(* Logix 5000 project; controller SRP_BullPMM_TestBench_V1 vendor 1 type 14 code 77 rev 20.11; software revision 20.05 *)

TASK MainTask (continuous, watchdog 500 ms) : MainProgram

MODULES
   Controller : vendor 1 type 14 code 77 (CompactLogixL32EController 0, rev 20.11)
      LocalENB : 1769-L32E Ethernet Port (CompactLogixL32Ethernet 1, rev 20.11)
         VSD_DC : vendor 1 type 123 code 121 (Ethernet 192.168.2.130, rev 5.6, Output RPI 20 ms)
             : vendor 1 type 123 code 8192 (DPI 5, rev 4.1)
      Local : CompactBus (CompactVirtualAdapter 3, rev 20.11)
END_MODULES

VAR_GLOBAL   (* controller tags *)
   CTU_SRPSim : COUNTER := (PRE := 280, ACC := 248);
   CurrentLimitLocal : INT;
   DC_CommandOFF : BOOL;
   DC_CommandON : BOOL;
   DC_CommandReset : BOOL;
   DC_CommandSpeed : INT;
   DC_CurrentLimit : INT;
   DC_LoadSent : INT := 7;
   DC_MaxLoad : REAL := 15.0;
   DC_MinLoad : REAL := 3.0;
   DC_OutputPower : REAL;
   DC_OutputVoltage : REAL;
   DC_RPMFeedback : INT := -22;
   DC_RPMReference : DINT := 100;
   DC_SpeedReference : INT := 140;
   DC_Timer_OFF : TIMER := (PRE := 1000);
   DC_Timer_ON : TIMER := (PRE := 1000);
   DC_Timer_RST : TIMER := (PRE := 1000);
   habilitado : BOOL; {access Read Only}
   Samples : INT := 280;
   SPM : REAL := 8.51;
   SRP_Displacement : REAL[400] := ([0] := 4.0, [1] := 1.0, [2] := 2.0, [3] := 3.0, [4] := 4.0, [5] := 5.0, [6] := 6.0, [7] := 7.0, [8] := 8.0, [9] := 9.0, [10] := 10.0, [11] := 11.0, [12] := 12.0, [13] := 13.0, [14] := 14.0, [15] := 15.0, [16] := 16.0, [17] := 17.0, [18] := 18.0, [19] := 19.0, [20] := 20.0, [21] := 21.0, [22] := 22.0, [23] := 23.0, [24] := 24.0, [25] := 25.0, [26] := 26.0, [27] := 27.0, [28] := 28.0, [29] := 29.0, [30] := 30.0, [31] := 31.0, [32] := 32.0, [33] := 33.0, [34] := 34.0, [35] := 35.0, [36] := 36.0, [37] := 37.0, [38] := 38.0, [39] := 39.0, [40] := 40.0, [41] := 41.0, [42] := 42.0, [43] := 43.0, [44] := 44.0, [45] := 45.0, [46] := 46.0, [47] := 47.0, [48] := 48.0, [49] := 49.0, [50] := 50.0, [51] := 51.0, [52] := 52.0, [53] := 53.0, [54] := 54.0, [55] := 55.0, [56] := 56.0, [57] := 57.0, [58] := 58.0, [59] := 59.0,
        [60] := 60.0, [61] := 61.0, [62] := 62.0, [63] := 63.0, [64] := 64.0, [65] := 65.0, [66] := 66.0, [67] := 67.0, [68] := 68.0, [69] := 69.0, [70] := 70.0, [71] := 71.0, [72] := 72.0, [73] := 73.0, [74] := 74.0, [75] := 75.0, [76] := 76.0, [77] := 77.0, [78] := 78.0, [79] := 79.0, [80] := 80.0, [81] := 81.0, [82] := 82.0, [83] := 83.0, [84] := 84.0, [85] := 85.0, [86] := 86.0, [87] := 87.0, [88] := 88.0, [89] := 89.0, [90] := 90.0, [91] := 91.0, [92] := 92.0, [93] := 93.0, [94] := 94.0, [95] := 95.0, [96] := 96.0, [97] := 97.0, [98] := 98.0, [99] := 99.0, [100] := 100.0, [101] := 101.0, [102] := 102.0, [103] := 103.0, [104] := 104.0, [105] := 105.0, [106] := 106.0, [107] := 107.0, [108] := 108.0, [109] := 109.0, [110] := 110.0, [111] := 111.0, [112] := 112.0, [113] := 113.0, [114] := 114.0, [115] := 115.0, [116] := 116.0, [117] := 117.0, [118] := 118.0, [119] := 119.0,
        [120] := 120.0, [121] := 121.0, [122] := 122.0, [123] := 123.0, [124] := 124.0, [125] := 125.0, [126] := 126.0, [127] := 127.0, [128] := 128.0, [129] := 129.0, [130] := 130.0, [131] := 131.0, [132] := 132.0, [133] := 133.0, [134] := 134.0, [135] := 135.0, [136] := 136.0, [137] := 137.0, [138] := 138.0, [139] := 139.0, [140] := 140.0); {access Read Only}
   SRP_Displacement_actual : REAL := 34.528854; {produced, access Read Only}
   SRP_Load : REAL[400] := ([1] := 12.0, [2] := 5.0, [3] := 6.0, [4] := 7.0, [5] := 89.0, [6] := 9.0, [7] := 3.0, [8] := 4.0, [9] := 6.0, [12] := 8.0, [14] := 56.0, [16] := 56.0, [18] := 56.0, [21] := 8765.0, [24] := 5678.0, [26] := 5678.0, [27] := 567.0, [28] := 8.0, [29] := 324.0, [31] := 234.0, [32] := 324.0, [33] := 234.0, [34] := 234.0, [35] := 342.0, [36] := 34.0, [43] := 432.0, [45] := 4.0, [46] := 4.0, [47] := 4.0, [48] := 4.0, [50] := 3.0, [52] := 2.0, [55] := 245.0, [56] := 2345.0, [57] := 2345.0, [58] := 724.0, [59] := 4325.0, [60] := 3245.0, [61] := 2345.0, [86] := 2345.0, [89] := 2345.0, [91] := 2345.0, [92] := 2345.0, [98] := 234.0, [99] := 4.0, [100] := 2.0, [101] := 3.0, [102] := 45.0, [103] := 2345.0, [104] := 2345.0, [105] := 5234.0, [106] := 354.0, [170] := 123.0, [191] := 345.0, [215] := 132.0, [216] := 5.0, [217] := 6.0, [219] := 8.0, [220] := 435.0, [221] := 34.0,
        [222] := 34.0, [223] := 3.0, [226] := 234.0, [227] := 3.0, [228] := 456.0, [231] := 546.0, [232] := 543.0, [233] := 453.0, [234] := 543.0, [235] := 34.0, [236] := 4.0, [294] := 4234.0, [295] := 3.0, [296] := 34.0, [297] := 4334.0, [298] := 34.0, [299] := 34.0, [300] := 43.0, [301] := 34.0, [303] := 1234.0); {access Read Only}
   SRP_Load_Actual : REAL := 8.460728; {produced, access Read Only}
   SRP_LoadEXC : REAL[400] := ([0] := 9.395175, [1] := 9.461731, [2] := 9.6614, [3] := 9.7812, [4] := 9.741267, [5] := 9.711983, [6] := 9.703996, [7] := 9.725293, [8] := 9.805161, [9] := 9.842433, [10] := 9.794512, [11] := 9.749254, [12] := 9.70932, [13] := 9.69601, [14] := 9.735943, [15] := 9.7306185, [16] := 9.634778, [17] := 9.586858, [18] := 9.634777, [19] := 9.751916, [20] := 10.007491, [21] := 10.223133, [22] := 10.358908, [23] := 10.473384, [24] := 10.545264, [25] := 10.633119, [26] := 10.752919, [27] := 10.856748, [28] := 10.928628, [29] := 11.029794, [30] := 11.109661, [31] := 11.220809, [32] := 11.347599, [33] := 11.419147, [34] := 11.463074, [35] := 11.515653, [36] := 11.572558, [37] := 11.655421, [38] := 11.751262, [39] := 11.805838, [40] := 11.839782, [41] := 11.900348, [42] := 11.974224, [43] := 11.940947, [44] := 11.854091, [45] := 11.73795, [46] := 11.607167, [47] := 11.4471, [48] := 11.27239, [49] := 11.15625, [50] := 11.069394, [51] := 10.976548, [52] := 10.880708, [53] := 10.774218, [54] := 10.662403, [55] := 10.571887, [56] := 10.492021, [57] := 10.393517, [58] := 10.321636, [59] := 10.257743,
        [60] := 10.193849, [61] := 10.105995, [62] := 10.018141, [63] := 9.930286, [64] := 9.842432, [65] := 9.762565, [66] := 9.682698, [67] := 9.634777, [68] := 9.586857, [69] := 9.706658, [70] := 9.826459, [71] := 9.938273, [72] := 10.050088, [73] := 10.082034, [74] := 10.113981, [75] := 10.177875, [76] := 10.241769, [77] := 10.321636, [78] := 10.401504, [79] := 10.409491, [80] := 10.417477, [81] := 10.409491, [82] := 10.401504, [83] := 10.457411, [84] := 10.518642, [85] := 10.534616, [86] := 10.529291, [87] := 10.481371, [88] := 10.476047, [89] := 10.555914, [90] := 10.63312, [91] := 10.705, [92] := 10.715649, [93] := 10.603834, [94] := 10.476047, [95] := 10.316312, [96] := 10.17255, [97] := 10.060737, [98] := 9.970221, [99] := 9.9223, [100] := 9.850419, [101] := 9.7306185, [102] := 9.608155, [103] := 9.480367, [104] := 9.397838, [105] := 9.405825, [106] := 9.405825, [107] := 9.389851, [108] := 9.34193, [109] := 9.230116, [110] := 9.131613, [111] := 9.059732, [112] := 9.049084, [113] := 9.10499, [114] := 9.08103, [115] := 9.017137, [116] := 8.9266205, [117] := 8.822793, [118] := 8.873376, [119] := 9.0011635,
        [120] := 9.155573, [121] := 9.323295, [122] := 9.427122, [123] := 9.499002, [124] := 9.549585, [125] := 9.589519, [126] := 9.682697, [127] := 9.802498, [128] := 9.906326, [129] := 10.002167, [130] := 10.012816, [131] := 9.980869, [132] := 9.980869, [133] := 9.996842, [134] := 9.986194, [135] := 9.962234, [136] := 9.980869, [137] := 10.0208025, [138] := 10.018141, [139] := 9.994181, [140] := 10.042101, [141] := 10.098008, [142] := 10.145928, [143] := 10.193849, [144] := 10.066061, [145] := 9.938273, [146] := 9.778539, [147] := 9.618804, [148] := 9.578871, [149] := 9.538937, [150] := 9.546924, [151] := 9.55491, [152] := 9.443096, [153] := 9.331282, [154] := 9.251414, [155] := 9.171547, [156] := 9.259401, [157] := 9.347255, [158] := 9.331282, [159] := 9.315308, [160] := 9.219467, [161] := 9.123626, [162] := 9.155573, [163] := 9.18752, [164] := 9.259401, [165] := 9.331282, [166] := 9.259401, [167] := 9.182196, [168] := 9.166222, [169] := 9.2168045, [170] := 9.400499, [171] := 9.565559, [172] := 9.693347, [173] := 9.762566, [174] := 9.714645, [175] := 9.688023, [176] := 9.703996, [177] := 9.746592, [178] := 9.842432, [179] := 9.901002,
        [180] := 9.885028, [181] := 9.834445, [182] := 9.714644, [183] := 9.634777, [184] := 9.634777, [185] := 9.640101, [186] := 9.656075, [187] := 9.624128, [188] := 9.496341, [189] := 9.37654, [190] := 9.272713, [191] := 9.184858, [192] := 9.128951, [193] := 9.046422, [194] := 8.910647, [195] := 8.665721, [196] := 8.434105, [197] := 8.223788, [198] := 8.02412, [199] := 7.936266, [200] := 7.904319, [201] := 7.851074, [202] := 7.78718, [203] := 7.6647167, [204] := 7.5129685, [205] := 7.398492, [206] := 7.302651, [207] := 7.281353, [208] := 7.2973266, [209] := 7.238757, [210] := 7.1429167, [211] := 6.993831, [212] := 6.8181233, [213] := 6.706309, [214] := 6.6264415, [215] := 6.6796865, [216] := 6.799487, [217] := 6.903315, [218] := 6.999156, [219] := 7.1056457, [220] := 7.2174597, [221] := 7.3771944, [222] := 7.622121, [223] := 7.773869, [224] := 7.925617, [225] := 7.91763, [226] := 7.909643, [227] := 7.909643, [228] := 7.909643, [229] := 8.077365, [230] := 8.245086, [231] := 8.300993, [232] := 8.3569, [233] := 8.340926, [234] := 8.324953, [235] := 8.460728, [236] := 8.596502, [237] := 8.70033, [238] := 8.804157, [239] := 8.79617,
        [240] := 8.788184, [241] := 8.788184, [242] := 8.788184, [243] := 8.77221, [244] := 8.756237, [245] := 8.588515, [246] := 8.420794, [247] := 8.38086, [248] := 8.340927, [249] := 8.412807, [250] := 8.468715, [251] := 8.420794, [252] := 8.399496, [253] := 8.431443, [254] := 8.476701, [255] := 8.548582, [256] := 8.580528, [257] := 8.532608, [258] := 8.497999, [259] := 8.490012, [260] := 8.503324, [261] := 8.559231, [262] := 8.591178, [263] := 8.575204, [264] := 8.56988, [265] := 8.585853, [266] := 8.631111, [267] := 8.734939, [268] := 8.84409, [269] := 8.963892, [270] := 9.081031, [271] := 9.192845, [272] := 9.278037, [273] := 9.309984, [274] := 9.325957, [275] := 9.309984, [276] := 9.363229, [277] := 9.554911, [278] := 9.618804, [279] := 9.682698);
   SRP_MaxPower : REAL := 28.520952;
   SRP_MinPower : REAL := -11.989768;
   SRP_PositionEXC : REAL[400] := ([1] := 0.0550175, [2] := 0.22007, [3] := 0.4084145, [4] := 0.643343, [5] := 0.8989175, [6] := 1.195784, [7] := 1.5143573, [8] := 1.8763443, [9] := 2.2604218, [10] := 2.6886797, [11] := 3.1391559, [12] := 3.6340683, [13] := 4.147569, [14] := 4.698246, [15] := 5.2654533, [16] := 5.865721, [17] := 6.4805126, [18] := 7.1243505, [19] := 7.78114, [20] := 8.463832, [21] := 9.158964, [22] := 9.878975, [23] := 10.613574, [24] := 11.377348, [25] := 12.155543, [26] := 12.962581, [27] := 13.778378, [28] := 14.611691, [29] := 15.740422, [30] := 16.600204, [31] := 17.481466, [32] := 18.373468, [33] := 19.2797, [34] := 20.193047, [35] := 21.118301, [36] := 22.049511, [37] := 22.99865, [38] := 23.956749, [39] := 24.928076, [40] := 25.906015, [41] := 26.89821, [42] := 27.897532, [43] := 28.908155, [44] := 29.92443, [45] := 30.958275, [46] := 32.000904, [47] := 33.057575, [48] := 34.121273, [49] := 35.193996, [50] := 36.271236, [51] := 37.35984, [52] := 38.454124, [53] := 39.561394, [54] := 40.67515, [55] := 41.798325, [56] := 42.926197, [57] := 44.44635, [58] := 45.59054, [59] := 46.757927, [60] := 47.925312,
        [61] := 49.113125, [62] := 50.300934, [63] := 51.439133, [64] := 52.57733, [65] := 53.71554, [66] := 54.853752, [67] := 56.007725, [68] := 57.161697, [69] := 58.29858, [70] := 59.435463, [71] := 60.54371, [72] := 61.651955, [73] := 62.754997, [74] := 63.858036, [75] := 64.96143, [76] := 66.06483, [77] := 67.1463, [78] := 68.22777, [79] := 69.277466, [80] := 70.327156, [81] := 71.36186, [82] := 72.39657, [83] := 73.41511, [84] := 74.763824, [85] := 75.75438, [86] := 76.731834, [87] := 77.68309, [88] := 78.62532, [89] := 79.54948, [90] := 80.46515, [91] := 81.36385, [92] := 82.25429, [93] := 83.1282, [94] := 83.99117, [95] := 84.8323, [96] := 85.65761, [97] := 86.45127, [98] := 87.23202, [99] := 87.98693, [100] := 88.73018, [101] := 89.45013, [102] := 90.154045, [103] := 90.82591, [104] := 91.48115, [105] := 92.103096, [106] := 92.711365, [107] := 93.29226, [108] := 93.858185, [109] := 94.39419, [110] := 94.9114, [111] := 95.391045, [112] := 96.00089, [113] := 96.43602, [114] := 96.84068, [115] := 97.23012, [116] := 97.581314, [117] := 97.91339, [118] := 98.21293, [119] := 98.4962, [120] := 98.7474,
        [121] := 98.98255, [122] := 99.18755, [123] := 99.37747, [124] := 99.53332, [125] := 99.672134, [126] := 99.77987, [127] := 99.87206, [128] := 99.935196, [129] := 99.983795, [130] := 99.99795, [131] := 99.99487, [132] := 99.96849, [133] := 99.93045, [134] := 99.8579, [135] := 99.76811, [136] := 99.64918, [137] := 99.51568, [138] := 99.35959, [139] := 99.1922, [140] := 98.93282, [141] := 98.72924, [142] := 98.49876, [143] := 98.26827, [144] := 98.00428, [145] := 97.74029, [146] := 97.44318, [147] := 97.14606, [148] := 96.822845, [149] := 96.499626, [150] := 96.147736, [151] := 95.795845, [152] := 95.40002, [153] := 95.004196, [154] := 94.58556, [155] := 94.16693, [156] := 93.73634, [157] := 93.305756, [158] := 92.83442, [159] := 92.36308, [160] := 91.870316, [161] := 91.377556, [162] := 90.877785, [163] := 90.37801, [164] := 89.84918, [165] := 89.32036, [166] := 88.761856, [167] := 88.01027, [168] := 87.43099, [169] := 86.84538, [170] := 86.2471, [171] := 85.63856, [172] := 85.00949, [173] := 84.37339, [174] := 83.723206, [175] := 83.06744, [176] := 82.400505, [177] := 81.722916, [178] := 81.02402, [179] := 80.31708, [180] := 79.59406,
        [181] := 78.86634, [182] := 78.12919, [183] := 77.38295, [184] := 76.61854, [185] := 75.84359, [186] := 75.04756, [187] := 74.24831, [188] := 73.44262, [189] := 72.63172, [190] := 71.8104, [191] := 70.97654, [192] := 70.117615, [193] := 69.25514, [194] := 68.385605, [195] := 67.223434, [196] := 66.349724, [197] := 65.45152, [198] := 64.541084, [199] := 63.614063, [200] := 62.67875, [201] := 61.744232, [202] := 60.810116, [203] := 59.862404, [204] := 58.907894, [205] := 57.93054, [206] := 56.94176, [207] := 55.949615, [208] := 54.955784, [209] := 53.960396, [210] := 52.964237, [211] := 51.950417, [212] := 50.92777, [213] := 49.88953, [214] := 48.843502, [215] := 47.795254, [216] := 46.7459, [217] := 45.690845, [218] := 44.632946, [219] := 43.56501, [220] := 42.49205, [221] := 41.413986, [222] := 39.97316, [223] := 38.891975, [224] := 37.810795, [225] := 36.722637, [226] := 35.634483, [227] := 34.528854, [228] := 33.423225, [229] := 32.329132, [230] := 31.23504, [231] := 30.155361, [232] := 29.075682, [233] := 27.987307, [234] := 26.898933, [235] := 25.821117, [236] := 24.743301, [237] := 23.68875, [238] := 22.634195, [239] := 21.607874, [240] := 20.581553,
        [241] := 19.584843, [242] := 18.588135, [243] := 17.632542, [244] := 16.676949, [245] := 15.761359, [246] := 14.84577, [247] := 13.965392, [248] := 13.085015, [249] := 12.251199, [250] := 11.154951, [251] := 10.367658, [252] := 9.596523, [253] := 8.857708, [254] := 8.136012, [255] := 7.4485517, [256] := 6.7788615, [257] := 6.144711, [258] := 5.529149, [259] := 4.950763, [260] := 4.3940463, [261] := 3.8806663, [262] := 3.3902075, [263] := 2.945591, [264] := 2.520764, [265] := 2.1355166, [266] := 1.7710685, [267] := 1.448219, [268] := 1.148738, [269] := 0.895994, [270] := 0.66532767, [271] := 0.47881666, [272] := 0.31461334, [273] := 0.19502534, [274] := 0.096083336, [275] := 0.038433332, [276] := 0.009929333, [277] := 0.03971733, [278] := 0.049646668, [279] := 0.059576);
   SRP_Power : REAL[400] := ([0] := 2.551885, [1] := 2.526211, [2] := 2.762145, [3] := 3.15088, [4] := 3.471027, [5] := 3.689743, [6] := 4.114319, [7] := 4.615038, [8] := 4.850739, [9] := 5.001896, [10] := 5.272432, [11] := 5.59496, [12] := 5.888859, [13] := 6.347629, [14] := 6.84288, [15] := 7.367318, [16] := 7.921212, [17] := 8.516989, [18] := 9.109633, [19] := 9.632602, [20] := 10.197533, [21] := 10.698328, [22] := 11.190563, [23] := 11.553818, [24] := 11.697866, [25] := 11.495567, [26] := 10.985658, [27] := 10.299884, [28] := 9.439834, [29] := 8.447996, [30] := 7.398052, [31] := 6.339027, [32] := 4.935925, [33] := 3.031238, [34] := 1.459401, [35] := 0.276735, [36] := -0.995331, [37] := -2.203813, [38] := -2.905728, [39] := -3.235214, [40] := -3.565211, [41] := -3.949811, [42] := -4.18803, [43] := -4.357996, [44] := -4.674874, [45] := -4.990204, [46] := -5.242468, [47] := -5.435884, [48] := -5.624201, [49] := -6.038198, [50] := -6.693041, [51] := -7.339044, [52] := -8.051254, [53] := -8.895816, [54] := -9.61421, [55] := -10.201138, [56] := -10.823343, [57] := -11.339426, [58] := -11.636271, [59] := -11.782147,
        [60] := -11.972128, [61] := -11.989768, [62] := -11.704662, [63] := -11.330022, [64] := -10.987564, [65] := -10.524297, [66] := -9.882706, [67] := -9.189292, [68] := -8.584183, [69] := -7.851256, [70] := -7.017601, [71] := -6.200305, [72] := -5.343426, [73] := -4.430933, [74] := -3.576711, [75] := -2.761184, [76] := -1.932628, [77] := -0.54998, [78] := 1.023285, [79] := 2.116259, [80] := 3.323442, [81] := 4.80824, [82] := 6.057144, [83] := 7.129545, [84] := 8.445454, [85] := 9.693588, [86] := 10.728734, [87] := 11.758366, [88] := 12.826331, [89] := 13.582999, [90] := 14.218866, [91] := 15.069524, [92] := 15.737838, [93] := 16.248062, [94] := 16.888288, [95] := 17.60809, [96] := 18.025164, [97] := 18.633614, [98] := 19.340208, [99] := 19.911589, [100] := 20.582422, [101] := 21.522118, [102] := 22.43875, [103] := 23.26365, [104] := 24.143408, [105] := 25.048727, [106] := 25.803514, [107] := 26.474516, [108] := 27.176193, [109] := 27.786386, [110] := 28.26233, [111] := 28.520952, [112] := 28.501911, [113] := 28.034796, [114] := 27.190903, [115] := 26.228785, [116] := 24.982784, [117] := 23.454718, [118] := 21.755957, [119] := 20.000027,
        [120] := 18.192253, [121] := 16.202557, [122] := 14.243646, [123] := 12.335317, [124] := 10.649885, [125] := 9.217575, [126] := 8.083941, [127] := 7.108335, [128] := 6.272891, [129] := 5.557211, [130] := 4.842691, [131] := 4.222987, [132] := 3.666158, [133] := 3.238251, [134] := 2.8715, [135] := 2.659773, [136] := 2.569013, [137] := 2.589529, [138] := 2.578462, [139] := 2.53984, [140] := 2.679924, [141] := 4.4444447);
   SRP_SimActualPower : REAL;
   SRP_SimActualStroke : DINT; {produced}
   SRP_Simulation : BOOL := 1;
   SRP_StrokeDetection : INT[400] := ([0] := 1, [1] := 1, [2] := 1, [3] := 1, [4] := 1, [5] := 1, [6] := 1);
   Test_TagExcel : INT := 141;
   Timer_SRPsim : TIMER := (PRE := 25, ACC := 23, EN := 1, TT := 1);
END_VAR

PROGRAM MainProgram   (* main routine MainRoutine *)
VAR
   SCL_01 : SCALE := (InRawMax := 28.520952, InRawMin := -11.989768, InEUMax := 15.0, InEUMin := 3.0, Out := 6.551584);
END_VAR

ROUTINE MainRoutine   (* ladder *)
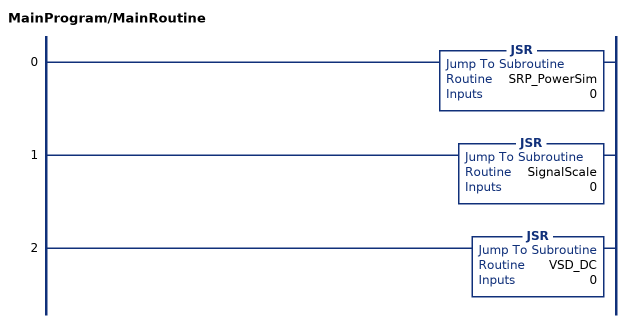
   0: JSR(SRP_PowerSim,0);
   1: JSR(SignalScale,0);
   2: JSR(VSD_DC,0);
END_ROUTINE

ROUTINE SignalScale   (* function block diagram *)
   SHEET 1
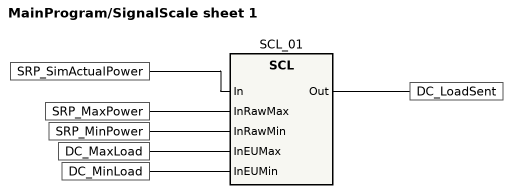
   SCL_01 : SCL(In := SRP_SimActualPower, InRawMax := SRP_MaxPower, InRawMin := SRP_MinPower, InEUMax := DC_MaxLoad, InEUMin := DC_MinLoad);
   DC_LoadSent := SCL_01.Out;
END_ROUTINE

ROUTINE SRP_PowerSim   (* ladder *)
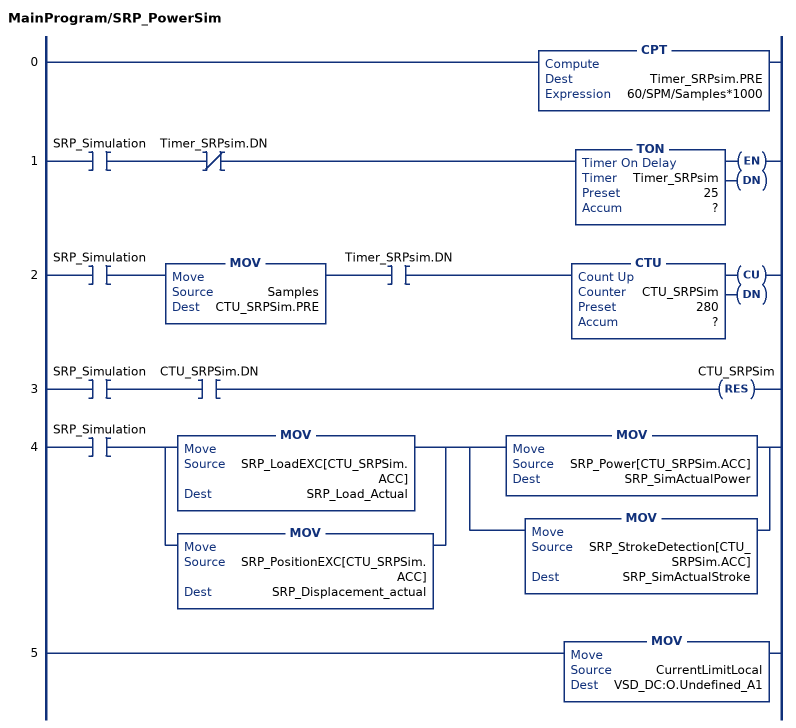
   0: CPT(Timer_SRPsim.PRE,60/SPM/Samples*1000);
   1: XIC(SRP_Simulation)XIO(Timer_SRPsim.DN)TON(Timer_SRPsim,?,?);
   2: XIC(SRP_Simulation)MOV(Samples,CTU_SRPSim.PRE)XIC(Timer_SRPsim.DN)CTU(CTU_SRPSim,?,?);
   3: XIC(SRP_Simulation)XIC(CTU_SRPSim.DN)RES(CTU_SRPSim);
   4: XIC(SRP_Simulation)[MOV(SRP_LoadEXC[CTU_SRPSim.ACC],SRP_Load_Actual) ,MOV(SRP_PositionEXC[CTU_SRPSim.ACC],SRP_Displacement_actual) ][MOV(SRP_Power[CTU_SRPSim.ACC],SRP_SimActualPower) ,MOV(SRP_StrokeDetection[CTU_SRPSim.ACC],SRP_SimActualStroke) ];
   5: MOV(CurrentLimitLocal,VSD_DC:O.Undefined_A1);
END_ROUTINE

ROUTINE VSD_DC   (* ladder *)
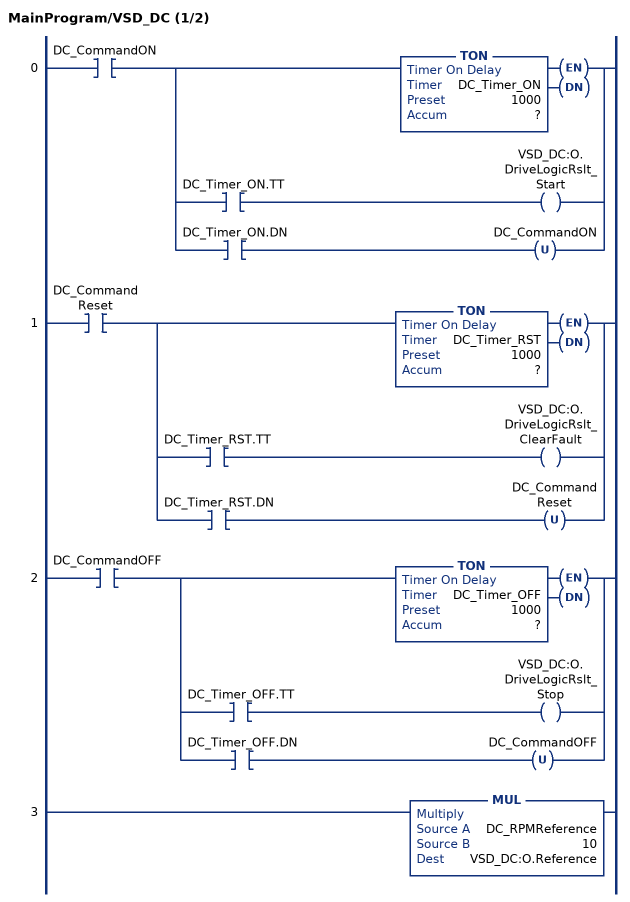
   0: XIC(DC_CommandON)[TON(DC_Timer_ON,?,?) ,[XIC(DC_Timer_ON.TT) OTE(VSD_DC:O.DriveLogicRslt_Start) ,XIC(DC_Timer_ON.DN) OTU(DC_CommandON) ] ];
   1: XIC(DC_CommandReset)[TON(DC_Timer_RST,?,?) ,[XIC(DC_Timer_RST.TT) OTE(VSD_DC:O.DriveLogicRslt_ClearFault) ,XIC(DC_Timer_RST.DN) OTU(DC_CommandReset) ] ];
   2: XIC(DC_CommandOFF)[TON(DC_Timer_OFF,?,?) ,[XIC(DC_Timer_OFF.TT) OTE(VSD_DC:O.DriveLogicRslt_Stop) ,XIC(DC_Timer_OFF.DN) OTU(DC_CommandOFF) ] ];
   3: MUL(DC_RPMReference,10,VSD_DC:O.Reference);
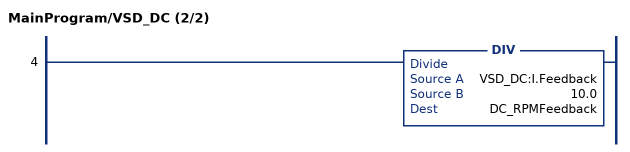
   4: DIV(VSD_DC:I.Feedback,10.0,DC_RPMFeedback);
END_ROUTINE
END_PROGRAM
